// TIA Portal V17 export
// export: Created 2023-12-22T15:05:25.562182Z, ExportSetting WithDefaults, DisplayName Totally Integrated Automation Portal, DisplayVersion V17, DisplayName TIA Portal Openness, DisplayVersion V17, DisplayName TIA Portal Version Control Interface, DisplayVersion V17, DisplayName STEP 7 Professional, DisplayVersion V17, DisplayName STEP 7 Safety, DisplayVersion V17, DisplayName WinCC Advanced, DisplayVersion V17
FUNCTION_BLOCK "Smena"   // FB17, LAD
{ S7_Optimized_Access := 'FALSE' }
VERSION : 0.1
// stored: AutoNumber true, IsIECCheckEnabled false, SetENOAutomatically false, UDAEnableTagReadback false
   VAR DB_SPECIFIC
      ON_1 : Struct
         Use : Bool;
         H : Int;
         "M" : Int;
      END_STRUCT;
      ON_2 : Struct
         Use : Bool;
         H : Int;
         "M" : Int;
      END_STRUCT;
      pos : Array[0..31] of Bool;
      Line_1 : Array[0..2] of Struct
         Water : Real;
         Reagent : Real;
      END_STRUCT;
      Line_2 : Array[0..2] of Struct
         Water : Real;
         Reagent : Real;
      END_STRUCT;
      "Time" : Array[0..2] of Struct
         Start_H : Int;
         Start_M : Int;
         "Date" : Int;
         Mounth : Int;
      END_STRUCT;
      Time_DTL : DTL;
   END_VAR
   VAR_TEMP
      x0 : Real;
      x1 : Real;
      x2 : Real;
      x3 : Real;
   END_VAR
   VAR_TEMP   // added for the SCL form of the ladder/FBD networks
      _w1 : Bool;
      _w2 : Bool;
   END_VAR
BEGIN

REGION Network 1: Первая запись
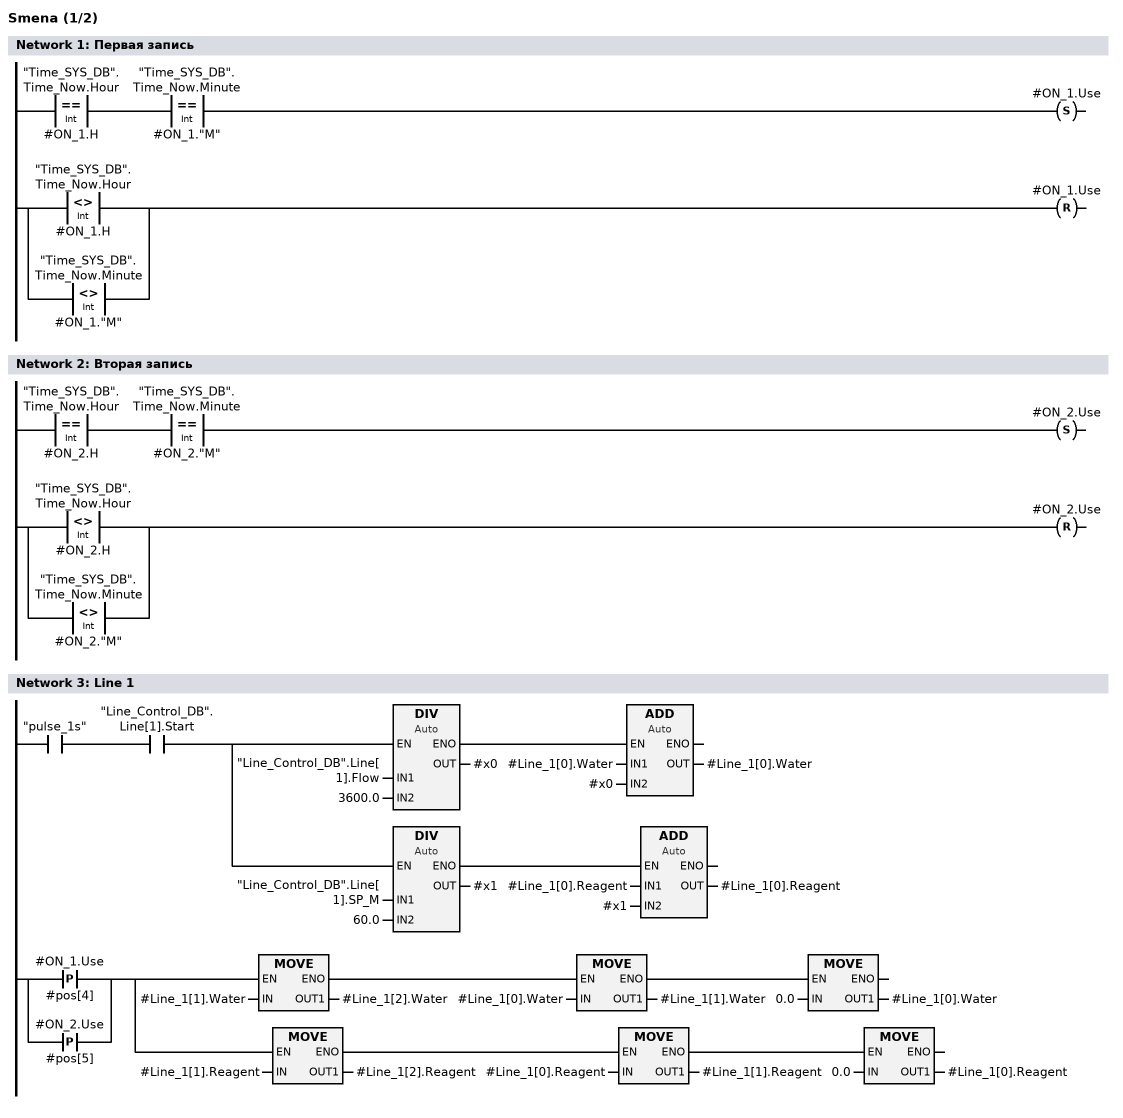
   RUNG wire#powerrail
      { S7_Templates := "SrcType := Int" } EQ_Contact(in1 := "Time_SYS_DB".Time_Now.Hour, in2 := #ON_1.H)
      { S7_Templates := "SrcType := Int" } EQ_Contact(in1 := "Time_SYS_DB".Time_Now.Minute, in2 := #ON_1."M")
      S_Coil( #ON_1.Use )
   END_RUNG
   RUNG wire#powerrail
      { S7_Templates := "SrcType := Int" } NE_Contact(in1 := "Time_SYS_DB".Time_Now.Hour, in2 := #ON_1.H)
      wire#w1
      R_Coil( #ON_1.Use )
   END_RUNG
   RUNG wire#powerrail
      { S7_Templates := "SrcType := Int" } NE_Contact(in1 := "Time_SYS_DB".Time_Now.Minute, in2 := #ON_1."M")
   END_RUNG wire#w1
   // the same network as SCL:
   IF ("Time_SYS_DB".Time_Now.Hour = #ON_1.H) AND ("Time_SYS_DB".Time_Now.Minute = #ON_1."M") THEN
       #ON_1.Use := TRUE;
   END_IF;
   IF ("Time_SYS_DB".Time_Now.Hour <> #ON_1.H) OR ("Time_SYS_DB".Time_Now.Minute <> #ON_1."M") THEN
       #ON_1.Use := FALSE;
   END_IF;
END_REGION

REGION Network 2: Вторая запись
   RUNG wire#powerrail
      { S7_Templates := "SrcType := Int" } EQ_Contact(in1 := "Time_SYS_DB".Time_Now.Hour, in2 := #ON_2.H)
      { S7_Templates := "SrcType := Int" } EQ_Contact(in1 := "Time_SYS_DB".Time_Now.Minute, in2 := #ON_2."M")
      S_Coil( #ON_2.Use )
   END_RUNG
   RUNG wire#powerrail
      { S7_Templates := "SrcType := Int" } NE_Contact(in1 := "Time_SYS_DB".Time_Now.Hour, in2 := #ON_2.H)
      wire#w1
      R_Coil( #ON_2.Use )
   END_RUNG
   RUNG wire#powerrail
      { S7_Templates := "SrcType := Int" } NE_Contact(in1 := "Time_SYS_DB".Time_Now.Minute, in2 := #ON_2."M")
   END_RUNG wire#w1
   // the same network as SCL:
   IF ("Time_SYS_DB".Time_Now.Hour = #ON_2.H) AND ("Time_SYS_DB".Time_Now.Minute = #ON_2."M") THEN
       #ON_2.Use := TRUE;
   END_IF;
   IF ("Time_SYS_DB".Time_Now.Hour <> #ON_2.H) OR ("Time_SYS_DB".Time_Now.Minute <> #ON_2."M") THEN
       #ON_2.Use := FALSE;
   END_IF;
END_REGION

REGION Network 3: Line 1
   RUNG wire#powerrail
      Contact( "pulse_1s" )
      Contact( "Line_Control_DB".Line[1].Start )
      wire#w1
      Div(in1 := "Line_Control_DB".Line[1].Flow, in2 := 3600.0, out => #x0)
      Add(in1 := #Line_1[0].Water, in2 := #x0, out => #Line_1[0].Water)
   END_RUNG
   RUNG wire#w1
      Div(in1 := "Line_Control_DB".Line[1].SP_M, in2 := 60.0, out => #x1)
      Add(in1 := #Line_1[0].Reagent, in2 := #x1, out => #Line_1[0].Reagent)
   END_RUNG
   RUNG wire#powerrail
      P_Contact(operand := #ON_1.Use, bit := #pos[4])
      wire#w2
      Move(in := #Line_1[1].Water, out1 => #Line_1[2].Water)
      Move(in := #Line_1[0].Water, out1 => #Line_1[1].Water)
      Move(in := 0.0, out1 => #Line_1[0].Water)
   END_RUNG
   RUNG wire#powerrail
      P_Contact(operand := #ON_2.Use, bit := #pos[5])
   END_RUNG wire#w2
   RUNG wire#w2
      Move(in := #Line_1[1].Reagent, out1 => #Line_1[2].Reagent)
      Move(in := #Line_1[0].Reagent, out1 => #Line_1[1].Reagent)
      Move(in := 0.0, out1 => #Line_1[0].Reagent)
   END_RUNG
   // the same network as SCL:
   IF "pulse_1s" AND "Line_Control_DB".Line[1].Start THEN
       #x0 := "Line_Control_DB".Line[1].Flow / 3600.0;
       #Line_1[0].Water := #Line_1[0].Water + #x0;
       #x1 := "Line_Control_DB".Line[1].SP_M / 60.0;
       #Line_1[0].Reagent := #Line_1[0].Reagent + #x1;
   END_IF;
   #_w1 := #ON_1.Use AND NOT #pos[4];   // rising edge of #ON_1.Use
   #pos[4] := #ON_1.Use;
   #_w2 := #ON_2.Use AND NOT #pos[5];   // rising edge of #ON_2.Use
   #pos[5] := #ON_2.Use;
   IF #_w1 OR #_w2 THEN
       #Line_1[2].Water := #Line_1[1].Water;
       #Line_1[1].Water := #Line_1[0].Water;
       #Line_1[0].Water := 0.0;
       #Line_1[2].Reagent := #Line_1[1].Reagent;
       #Line_1[1].Reagent := #Line_1[0].Reagent;
       #Line_1[0].Reagent := 0.0;
   END_IF;
END_REGION

REGION Network 4
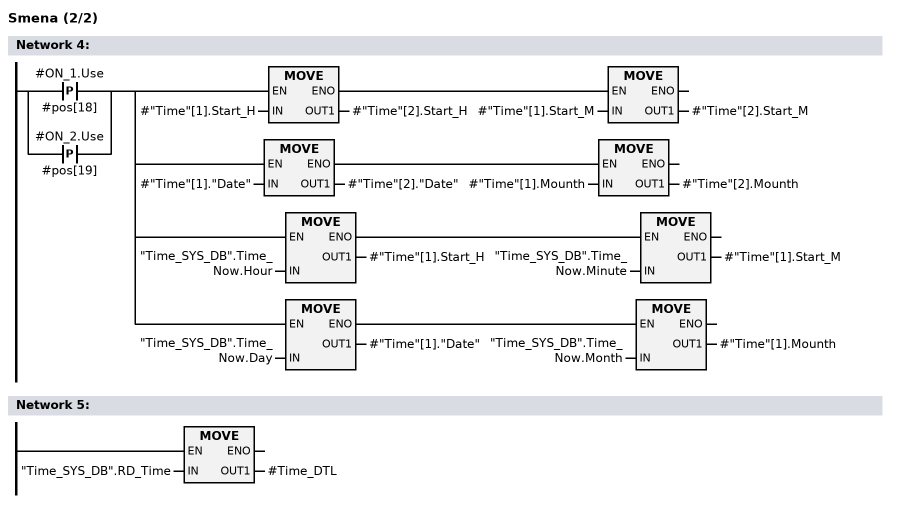
   RUNG wire#powerrail
      P_Contact(operand := #ON_1.Use, bit := #pos[18])
      wire#w1
      Move(in := #"Time"[1].Start_H, out1 => #"Time"[2].Start_H)
      Move(in := #"Time"[1].Start_M, out1 => #"Time"[2].Start_M)
   END_RUNG
   RUNG wire#powerrail
      P_Contact(operand := #ON_2.Use, bit := #pos[19])
   END_RUNG wire#w1
   RUNG wire#w1
      Move(in := #"Time"[1]."Date", out1 => #"Time"[2]."Date")
      Move(in := #"Time"[1].Mounth, out1 => #"Time"[2].Mounth)
   END_RUNG
   RUNG wire#w1
      Move(in := "Time_SYS_DB".Time_Now.Hour, out1 => #"Time"[1].Start_H)
      Move(in := "Time_SYS_DB".Time_Now.Minute, out1 => #"Time"[1].Start_M)
   END_RUNG
   RUNG wire#w1
      Move(in := "Time_SYS_DB".Time_Now.Day, out1 => #"Time"[1]."Date")
      Move(in := "Time_SYS_DB".Time_Now.Month, out1 => #"Time"[1].Mounth)
   END_RUNG
   // the same network as SCL:
   #_w1 := #ON_1.Use AND NOT #pos[18];   // rising edge of #ON_1.Use
   #pos[18] := #ON_1.Use;
   #_w2 := #ON_2.Use AND NOT #pos[19];   // rising edge of #ON_2.Use
   #pos[19] := #ON_2.Use;
   IF #_w1 OR #_w2 THEN
       #"Time"[2].Start_H := #"Time"[1].Start_H;
       #"Time"[2].Start_M := #"Time"[1].Start_M;
       #"Time"[2]."Date" := #"Time"[1]."Date";
       #"Time"[2].Mounth := #"Time"[1].Mounth;
       #"Time"[1].Start_H := "Time_SYS_DB".Time_Now.Hour;
       #"Time"[1].Start_M := "Time_SYS_DB".Time_Now.Minute;
       #"Time"[1]."Date" := "Time_SYS_DB".Time_Now.Day;
       #"Time"[1].Mounth := "Time_SYS_DB".Time_Now.Month;
   END_IF;
END_REGION

REGION Network 5
   RUNG wire#powerrail
      Move(in := "Time_SYS_DB".RD_Time, out1 => #Time_DTL)
   END_RUNG
   // the same network as SCL:
   #Time_DTL := "Time_SYS_DB".RD_Time;
END_REGION
END_FUNCTION_BLOCK
